(* PLC project Tc2_Utilities.F_TranslateFileTime64Bias Demo, tc3-libraries-kb TwinCAT 3.1 *)
(* stored: creationDateTime 2026-05-10T12:00:00, modificationDateTime 2026-05-10T12:00:00 *)

PROGRAM P_Demo_F_TranslateFileTime64Bias
  VAR
    rResult : T_FILETIME64;  (* F_TranslateFileTime64Bias 的返回值 *)
    bRun : BOOL;  (* 触发一次调用 *)
    ftIn : T_FILETIME64;  (* 测试用本地变量 *)
  END_VAR

            // ============================================================
// Tc2_Utilities.F_TranslateFileTime64Bias 演示程序（FUNCTION）
// ============================================================
// 验证步骤：
//   1. 引用 Tc2_Utilities（及类型所在依赖库 Tc2_System / Tc2_Standard）
//   2. 编译 + 登录
//   3. 强制 bRun := TRUE 一个周期
//   4. 观察 rResult 应为 对应本地时 11:00 的 FILETIME
// ============================================================

ftIn := DT_TO_FILETIME64(DT#2024-07-15-10:00:00);
IF bRun THEN
    rResult := F_TranslateFileTime64Bias(ftIn, 60, FALSE);
    bRun := FALSE;
END_IF;

          
END_PROGRAM
